// TIA Portal V19 export
VAR_GLOBAL   // PLC tag table "TT - General"
   iDkStart_S2 AT %I0.0 : Bool;   // NO
   iDkStop_S3 AT %I0.1 : Bool;   // NC
   iSelSchMan_Q2 AT %I0.2 : Bool;
   iDkReset_S4 AT %I0.3 : Bool;   // NO (reset VR)
   iStsNoodstop_S1 AT %I2.7 : Bool;   // NO
   oLmpAlarm_H1 AT %Q0.0 : Bool;
   oLmpWarningLowMaterial_H2 AT %Q1.7 : Bool;
   iSenPressure AT %I2.6 : Bool;   // true when pressure
END_VAR
